{attribute 'qualified_only'}
VAR_GLOBAL CONSTANT
    COMPONENT_BASE_ALARM_COUNT : UINT := 2;
END_VAR

(* stored: Version 1.1.0.1, ProductVersion 3.1.4024.12
   GVL Parameters_BaseComponent: Id {aeed3e49-fd03-4249-88b3-2d92a04d6e6b}, ParameterList True *)
